// TwinCAT 3 PLC project RK_PapestraatV01
// ProgramVersion: 3.1.4024.12
// libraries:
//   Tc2_Standard, * (Beckhoff Automation GmbH)
//   Tc2_System, * (Beckhoff Automation GmbH)
//   Tc3_Module, * (Beckhoff Automation GmbH)
//   VisuSymbols,3.5.10.0,System
// project tree:
//   / GlobalTextList.TcGTLO, PlcTask.TcTTO, Visualization Manager.TcVMO (not stored)
//   GVLs/ GVL.TcGVL
//   POUs/ fbLightControl.TcPOU, fbLightControlV2.TcPOU, fbLightControl_ButtonAndDetect.TcPOU, fbVerwarming.TcPOU, MAIN.TcPOU, SturingVerwarming.TcPOU
//   VISUs/ InitSoftware.TcVIS
// real-time tasks:
//   TASK PlcTask: cycle T#10ms, priority 20, ADS port 350
// I/O:
//   DEVICE Device 2 (EtherCAT), AmsNetId 5.83.127.149.3.1
//     Term 8 (EK1200) [EK1200-5000 EtherCAT Power supply (2A E-Bus)]
//       Term 7 (EL1809) [EL1809 16Ch. Dig. Input 24V, 3ms]
//       Term 8 (EL1809) [EL1809 16Ch. Dig. Input 24V, 3ms]
//       Term 9 (EL2809) [EL2809 16Ch. Dig. Output 24V, 0.5A]
//       Term 10 (EL1859) [EL1859 8Ch. Dig. Input 24V, 3ms, 8Ch. Dig. Output 24V, 0.5A]
//       Term 11 (EL1008) [EL1008 8Ch. Dig. Input 24V, 3ms]
//       Term 14 (EL2008) [EL2008 8Ch. Dig. Output 24V, 0.5A]
//       Term 15 (EL9011) [EL9011 End Terminal]
// variable links:
//   RK-PapestraatV01/RK-PapestraatV01 Instance <-> Device 2 (EtherCAT)/Term 8 (EK1200)/Term 10 (EL1859)
//     PlcTask Inputs/GVL.I_Input{32..39} <-> Channel {1..8}/Input  (8 links)
//     PlcTask Outputs/GVL.Q_Light{16..19} <-> Channel {9..12}/Output  (4 links)
//     PlcTask Outputs/SturingVerwarming.bBranderAan <-> Channel 13/Output
//     PlcTask Outputs/SturingVerwarming.bKlepBureau <-> Channel 16/Output
//     PlcTask Outputs/SturingVerwarming.bKlepGroteZaal <-> Channel 14/Output
//     PlcTask Outputs/SturingVerwarming.bKlepKleineZaal <-> Channel 15/Output
//   RK-PapestraatV01/RK-PapestraatV01 Instance <-> Device 2 (EtherCAT)/Term 8 (EK1200)/Term 11 (EL1008)
//     PlcTask Inputs/SturingVerwarming.bDrukknopBureau <-> Channel 5/Input
//     PlcTask Inputs/SturingVerwarming.bDrukknopGroteZaal <-> Channel 1/Input
//     PlcTask Inputs/SturingVerwarming.bDrukknopKleineZaal <-> Channel 3/Input
//   RK-PapestraatV01/RK-PapestraatV01 Instance <-> Device 2 (EtherCAT)/Term 8 (EK1200)/Term 14 (EL2008)
//     PlcTask Outputs/SturingVerwarming.bKlepBureau <-> Channel 5/Output
//     PlcTask Outputs/SturingVerwarming.bKlepGroteZaal <-> Channel 1/Output
//     PlcTask Outputs/SturingVerwarming.bKlepKleineZaal <-> Channel 3/Output
//   RK-PapestraatV01/RK-PapestraatV01 Instance <-> Device 2 (EtherCAT)/Term 8 (EK1200)/Term 7 (EL1809)
//     PlcTask Inputs/GVL.I_Input01 <-> Channel 2/Input
//     PlcTask Inputs/GVL.I_Input02 <-> Channel 3/Input
//     PlcTask Inputs/GVL.I_Input03 <-> Channel 4/Input
//     PlcTask Inputs/GVL.I_Input04 <-> Channel 5/Input
//     PlcTask Inputs/GVL.I_Input05 <-> Channel 6/Input
//     PlcTask Inputs/GVL.I_Input06 <-> Channel 7/Input
//     PlcTask Inputs/GVL.I_Input08 <-> Channel 9/Input
//     PlcTask Inputs/GVL.I_Input09 <-> Channel 10/Input
//     PlcTask Inputs/GVL.I_Input10 <-> Channel 11/Input
//     PlcTask Inputs/GVL.I_Input11 <-> Channel 12/Input
//     PlcTask Inputs/GVL.I_Input12 <-> Channel 13/Input
//     PlcTask Inputs/GVL.I_Input13 <-> Channel 14/Input
//     PlcTask Inputs/GVL.I_Input14 <-> Channel 15/Input
//     PlcTask Inputs/GVL.I_Input15 <-> Channel 16/Input
//     PlcTask Inputs/SturingVerwarming.bThermostaatBureau <-> Channel 1/Input
//     PlcTask Inputs/SturingVerwarming.bThermostaatGroteZaal <-> Channel 8/Input
//   RK-PapestraatV01/RK-PapestraatV01 Instance <-> Device 2 (EtherCAT)/Term 8 (EK1200)/Term 8 (EL1809)
//     PlcTask Inputs/GVL.I_Input16 <-> Channel 1/Input
//     PlcTask Inputs/GVL.I_Input17 <-> Channel 2/Input
//     PlcTask Inputs/GVL.I_Input18 <-> Channel 3/Input
//     PlcTask Inputs/GVL.I_Input19 <-> Channel 4/Input
//     PlcTask Inputs/GVL.I_Input21 <-> Channel 6/Input
//     PlcTask Inputs/GVL.I_Input22 <-> Channel 7/Input
//     PlcTask Inputs/GVL.I_Input23 <-> Channel 8/Input
//     PlcTask Inputs/GVL.I_Input24 <-> Channel 9/Input
//     PlcTask Inputs/GVL.I_Input25 <-> Channel 10/Input
//     PlcTask Inputs/GVL.I_Input26 <-> Channel 11/Input
//     PlcTask Inputs/GVL.I_Input27 <-> Channel 12/Input
//     PlcTask Inputs/GVL.I_Input28 <-> Channel 13/Input
//     PlcTask Inputs/GVL.I_Input29 <-> Channel 14/Input
//     PlcTask Inputs/GVL.I_Input30 <-> Channel 15/Input
//     PlcTask Inputs/GVL.I_Input31 <-> Channel 16/Input
//     PlcTask Inputs/SturingVerwarming.bThermostaatKleineZaal <-> Channel 5/Input
//   RK-PapestraatV01/RK-PapestraatV01 Instance <-> Device 2 (EtherCAT)/Term 8 (EK1200)/Term 9 (EL2809)
//     PlcTask Outputs/GVL.Q_Light00 <-> Channel 1/Output
//     PlcTask Outputs/GVL.Q_Light01 <-> Channel 2/Output
//     PlcTask Outputs/GVL.Q_Light02 <-> Channel 3/Output
//     PlcTask Outputs/GVL.Q_Light03 <-> Channel 4/Output
//     PlcTask Outputs/GVL.Q_Light04 <-> Channel 5/Output
//     PlcTask Outputs/GVL.Q_Light05 <-> Channel 6/Output
//     PlcTask Outputs/GVL.Q_Light06 <-> Channel 7/Output
//     PlcTask Outputs/GVL.Q_Light07 <-> Channel 8/Output
//     PlcTask Outputs/GVL.Q_Light08 <-> Channel 9/Output
//     PlcTask Outputs/GVL.Q_Light09 <-> Channel 10/Output
//     PlcTask Outputs/GVL.Q_Light10 <-> Channel 11/Output
//     PlcTask Outputs/GVL.Q_Light11 <-> Channel 12/Output
//     PlcTask Outputs/GVL.Q_Light12 <-> Channel 13/Output
//     PlcTask Outputs/GVL.Q_Light13 <-> Channel 14/Output
//     PlcTask Outputs/GVL.Q_Light14 <-> Channel 15/Output
//     PlcTask Outputs/GVL.Q_Light15 <-> Channel 16/Output

CONFIGURATION RK_PapestraatV01
    RESOURCE PLC ON TwinCAT3
        TASK PlcTask(INTERVAL := T#10ms, PRIORITY := 20);
        PROGRAM MAIN WITH PlcTask : MAIN;
    END_RESOURCE
END_CONFIGURATION

// ---- GVLs/GVL.TcGVL
{attribute 'qualified_only'}
VAR_GLOBAL
	I_Input00		AT %I* :BOOL; // Thermostaat Bureau
	I_Input01		AT %I* :BOOL; // Ingang Bureau
	I_Input02		AT %I* :BOOL; // ingang Lesruimte Rechts
	I_Input03		AT %I* :BOOL; // ingang Lesruimte Links
	I_Input04		AT %I* :BOOL; // Voorbereiding knop uitgang
	I_Input05		AT %I* :BOOL; // Gang GarageZijde
	I_Input06		AT %I* :BOOL; // Knop Aan Trap (nog te ontdubbelen
	I_Input07		AT %I* :BOOL; // Thermostaat lesruimte
	I_Input08		AT %I* :BOOL; // lesruimte naar garage
	I_Input09		AT %I* :BOOL; // WC midden
	I_Input10		AT %I* :BOOL; // WC naast Tech
	I_Input11		AT %I* :BOOL; // Gang 1
	I_Input12		AT %I* :BOOL; // Gang 2
	I_Input13		AT %I* :BOOL; // Grote WC
	I_Input14		AT %I* :BOOL; // Tech Ruimte 
	I_Input15		AT %I* :BOOL; // opleidingslokaal rechts voorraan

	I_Input16		AT %I* :BOOL; // Lesruimte naar buiten
	I_Input17		AT %I* :BOOL; // AllesUitVoordeur
	I_Input18		AT %I* :BOOL; // 2de schakelaar opleidinslokaal deur naar berging
	I_Input19		AT %I* :BOOL; // Grime Grote WC
	I_Input20		AT %I* :BOOL; // Thermostaat vergader 
	I_Input21		AT %I* :BOOL; // c vergaderzaal
	I_Input22		AT %I* :BOOL; // Vergaderzaal DeurNaarBuiten 
	I_Input23		AT %I* :BOOL; // X Keuken
	I_Input24		AT %I* :BOOL; // Alles Uit 
	I_Input25		AT %I* :BOOL; // Garagezonder Deur Onderlinks
	I_Input26		AT %I* :BOOL; // Garagezonder Deur OnderRechts
	I_Input27		AT %I* :BOOL; // Poort 2 DeurDicht
	I_Input28		AT %I* :BOOL; // Poort 2 DeurOpen (Niet gebruikt)
	I_Input29		AT %I* :BOOL; // Poort 1 DeurDicht 
	I_Input30		AT %I* :BOOL; // Poort 1 DeurOpen (Niet Gebruikt)
	I_Input31		AT %I* :BOOL; // I ( opleiding deur naar buiten

	I_Input32		AT %I* :BOOL; // Garage drukknop
	I_Input33		AT %I* :BOOL; // Garage Drukknop2
	I_Input34		AT %I* :BOOL; // Verdieping 1 druknop 2
	I_Input35		AT %I* :BOOL; // AllesUit
	I_Input36		AT %I* :BOOL; // 
	I_Input37		AT %I* :BOOL;
	I_Input38		AT %I* :BOOL;
	I_Input39		AT %I* :BOOL;
	
//output values
	Q_Light00		AT %Q* :BOOL;	// Groot WC
	Q_Light01		AT %Q* :BOOL;	// Midden WC
	Q_Light02		AT %Q* :BOOL;   // Keuken
	Q_Light03		AT %Q* :BOOL;	// Buitenlicht achter
	Q_Light04		AT %Q* :BOOL;	// WC naast Tech Ruimte 
	Q_Light05		AT %Q* :BOOL;  	// vergaderzaal
	Q_Light06		AT %Q* :BOOL;  	// bureau
	Q_Light07		AT %Q* :BOOL;  	// Lesruimte deel 1
	Q_Light08		AT %Q* :BOOL;  	// Garage Deur	
	Q_Light09		AT %Q* :BOOL;	// Garage enkel poort
	Q_Light10		AT %Q* :BOOL; 	// Verdiep 1 trap
	Q_Light11		AT %Q* :BOOL; 	// verdiep 1 ver
	Q_Light12		AT %Q* :BOOL;	// Berg Ruimte 
	Q_Light13		AT %Q* :BOOL;	// Gang Deel 2
	Q_Light14		AT %Q* :BOOL;	// GrimeLicht grote WC
	Q_Light15		AT %Q* :BOOL;	// Tech Ruimte
	
	Q_Light16		AT %Q* :BOOL;	// IndicatieLicht DeurGarage
	Q_Light17		AT %Q* :BOOL; 	// Lesruimte Deel 2
	Q_Light18		AT %Q* :BOOL; 	//
	Q_Light19		AT %Q* :BOOL;	// Lichtje GarageZonderDeur
	Q_Light20		AT %Q* :BOOL;	// Verwarming 1
	Q_Light21		AT %Q* :BOOL;	// Verwarming 2
	Q_Light22		AT %Q* :BOOL;	// Verwarming 3
	Q_Light23		AT %Q* :BOOL;	// Verwarming 4 
	
	
	LesruimteLichtAan		:BOOL;
	BureauLichtAan			:BOOL;
	Vergaderzaal			:BOOL;
	
// placeholder values
	I_Inputxx		AT %I* :BOOL;
	Q_LightXX		AT %Q* :BOOL;
	
	//I_Temp01		AT %I* :BOOL;
	//I_Temp02		AT %I* :BOOL;
	//I_Temp03		AT %I* :BOOL;
	//I_Temp04		AT %I* :BOOL;

	
END_VAR

// ---- POUs/MAIN.TcPOU
PROGRAM MAIN
VAR
	cnt			: UINT;
	
	fbLight00		: fbLightControl;
	fbLight01		: fbLightControl;
	fbLight02		: fbLightControl;
	fbLight03		: fbLightControl;
	fbLight04		: fbLightControl;
	fbLight05		: fbLightControl; // testje
	fbLight06		: fbLightControl;
	fbLight07		: fbLightControlV2;
	fbLight08		: fbLightControl_ButtonAndDetect;
	fbLight09		: fbLightControl;
	fbLight10		: fbLightControl;
	fbLight11		: fbLightControl;
	fbLight12		: fbLightControl;
	fbLight13		: fbLightControl;
	fbLight14		: fbLightControl;
//	fbLight15		: fbLightControl;
	
	bOutputActief	: BOOL;
	
	bForceOff		:BOOL;
	bForceOn		:BOOL;
	
	InputTriggerAllesUit		: R_trig; 
	
	LesruimteLichtAan: INT;
END_VAR

 cnt := cnt +1;



InputTriggerAllesUit(CLK := GVL.I_Input35 OR GVL.I_Input24 OR gvl.I_Input17);
	
// Actual light control

fbLight00(bButton:= GVL.I_Input32 , 
			bForceOff:= InputTriggerAllesUit.Q, 
			bForceOn:= , 
			bLight=> gvl.Q_Light07,
			bLight=> gvl.Q_Light04,
			);
// Grote WC hoofdlicht

GVL.Q_Light01 := GVL.I_Input09; //midden WC
GVL.Q_Light00 := GVL.I_Input13; // Grote WC 
GVL.Q_Light04 := GVL.I_Input10;// WC naast tech
GVL.Q_Light15 := GVL.I_Input14; // tech ruimte
GVL.Q_Light12 := GVL.I_Input08;// BergRuimte =Detector
GVL.Q_Light13 := GVL.I_Input11 OR GVL.I_Input12;// Gang deel2 detector


//verlichting Bureau
		


		

		
		// Licht Keuken
fbLight02(bButton:= GVL.I_Input03 OR GVL.I_Input23 ,  // check other button 
			bForceOff:= InputTriggerAllesUit.Q, 
			bForceOn:= , 
			bLight=> gvl.Q_Light02,
		);
		
// Licht Buiten	
fbLight03(bButton:= GVL.I_Input04 OR GVL.I_Input31 OR GVL.I_Input22, 
			bForceOff:= InputTriggerAllesUit.Q, 
			bForceOn:= , 
			bLight=> gvl.Q_Light03,
		);
		
// 	vergaderzaal

fbLight05(bButton:= GVL.I_Input21, 
			bForceOff:= InputTriggerAllesUit.Q, 
			bForceOn:= , 
			bLight=> gvl.Q_Light05
		);	
// Bureau

fbLight06(bButton:= GVL.I_Input01,
			bForceOff:= InputTriggerAllesUit.Q, 
			bForceOn:= , 
			
			bLight=> gvl.Q_Light06
		);	
// Lesruimte 	
fbLight07(bButtonhoofdFunctie:= GVL.I_Input02 OR GVL.I_Input15 ,
			bButton2 := GVL.I_Input18 OR GVL.I_Input16, // 16 should move to outside
			bForceOff:= InputTriggerAllesUit.Q, 
			bForceOn:= , 
			bLight1=> gvl.Q_Light07,
			bLight2=> gvl.Q_Light17
		);	
// Garage 	
fbLight08(bButton:= GVL.I_Input33 OR GVL.I_Input05 OR GVL.I_Input32 OR GVL.I_Input26,
			bDetection := GVL.I_Input37  ,
			bDeurDetectie :=  NOT(GVL.I_Input29) OR NOT(GVL.I_Input27),
			bForceOff:= InputTriggerAllesUit.Q, 
			bForceOn:= , 
			bInhibit:= InputTriggerAllesUit.Q, 
			bLight=> gvl.Q_Light08,
			bLight=> gvl.Q_Light09,
		);
// Deze knop laat toe om de detectie over te nemen 
// Logica nog te verbeteren met de alles uit samen te werken


(*TODO: remove after logic validation
gvl.Q_Light08 := gvl.Q_Light08 OR GVL.I_Input37;
gvl.Q_Light09 := gvl.Q_Light09 OR GVL.I_Input37;*)

// zaal boven
fbLight10(bButton:= GVL.I_Input34 OR GVL.I_Input06 OR GVL.I_Input25, 
			bForceOff:= InputTriggerAllesUit.Q, 
			bForceOn:= , 
			bLight=> gvl.Q_Light10,
			bLight=> gvl.Q_Light11
			);

// GrimeLicht Grote WC
fbLight14(bButton:= GVL.I_Input19 , 
			bForceOff:= InputTriggerAllesUit.Q, 
			bForceOn:= , 
			bLight=> gvl.Q_Light14
		);	

		
bOutputActief := fbLight00.bLight
				OR fbLight01.bLight
				OR fbLight02.bLight
				OR fbLight03.bLight
				OR fbLight04.bLight
				OR fbLight05.bLight
				OR fbLight06.bLight
				OR fbLight07.bLight1 OR fbLight07.bLight2
				OR fbLight08.bLight
				OR fbLight09.bLight
				OR fbLight10.bLight
				OR fbLight11.bLight
				OR fbLight12.bLight
				OR fbLight13.bLight
				OR fbLight14.bLight;

GVL.Q_Light16 :=  bOutputActief;				

// Activeer Verwarming

	GVL.LesruimteLichtAan := gvl.Q_Light07 OR gvl.Q_Light17 OR gvl.Q_Light02;
	GVL.BureauLichtAan	  := gvl.Q_Light06 ;
	GVL.Vergaderzaal	  := gvl.Q_Light05 ;

SturingVerwarming();

END_PROGRAM

// ---- POUs/fbLightControl.TcPOU
FUNCTION_BLOCK fbLightControl
		
VAR_INPUT
	bButton				: BOOL;
	bForceOff			: BOOL;
	bForceOn			: BOOL;

END_VAR
VAR_OUTPUT
	bLight				: BOOL;
	
END_VAR
VAR
	InputTrigger		: R_trig; 

	
END_VAR

// This is the first version, ignoring all debounce timers and other issues 
// Base function is a to allow switching a light on and of and having a general reset and general on ( used for construcion)

InputTrigger(CLK :=  bButton);

IF InputTrigger.Q THEN
	
	bLight := NOT(bLight);

END_IF

// Deze functie zorgt voor alles aan/Uit Functionaliteit
IF bForceOff THEN
	bLight := FALSE;
END_IF

IF bForceOn THEN
	bLight := TRUE;
END_IF

(*function notes: long klick functionality not added, most likley this will be part of another function
This could be a dedicated filter function linked to these functions as needed
*)

END_FUNCTION_BLOCK

// ---- POUs/fbLightControlV2.TcPOU
FUNCTION_BLOCK fbLightControlV2
		
VAR_INPUT
	bButtonhoofdFunctie				: BOOL;
	bButton2				: BOOL;
	bForceOff			: BOOL;
	bForceOn			: BOOL;

END_VAR
VAR_OUTPUT
	bLight1				: BOOL;
	bLight2				: BOOL;	
	
END_VAR
VAR
	InputTriggerHoofd		: R_trig; 
	InputTrigger2		: R_trig; 
	test:BOOL;
	iCaseVar			:UINT; 
	

	
END_VAR


// This is the first version, ignoring all debounce timers and other issues 
// Base function is a to allow switching a light on and of and having a general reset and general on ( used for construcion)

InputTriggerHoofd(CLK :=  bButtonhoofdFunctie);
InputTrigger2(CLK :=  bButton2);


IF InputTriggerHoofd.Q THEN
	
// ALs alles uit, dan alles aan
	IF (iCaseVar = 0) THEN
		iCaseVar := 1;
	ELSE
		iCaseVar := 0;
	END_IF
END_IF 

IF InputTrigger2.Q THEN
	
	// ALs alles aan, dan de voorste lichten uit
	IF (iCaseVar = 1) THEN
		iCaseVar := 2;
	ELSIF (iCaseVar = 2) THEN
		iCaseVar := 1;
	END_IF
	
END_IF

CASE iCaseVar OF
0:
    bLight1 := FALSE;
	bLight2 := FALSE;
1:
    bLight1 := TRUE;
	bLight2 := TRUE;	
2:
    bLight1 := TRUE;
	bLight2 := FALSE;
3: // eigenlijk niet noodzakelijk
	iCaseVar := 0;
ELSE
	iCaseVar := 0;
END_CASE;




// Deze functie zorgt voor alles aan/Uit Functionaliteit
IF bForceOff THEN
	iCaseVar := 0;
END_IF

IF bForceOn THEN
	iCaseVar := 1;
END_IF

(*function notes: long klick functionality not added, most likley this will be part of another function
This could be a dedicated filter function linked to these functions as needed
*)

END_FUNCTION_BLOCK

// ---- POUs/fbLightControl_ButtonAndDetect.TcPOU
FUNCTION_BLOCK fbLightControl_ButtonAndDetect
		
VAR_INPUT
	bButton				: BOOL;
	bDeurDetectie		: BOOL;
	bForceOff			: BOOL;
	bForceOn			: BOOL;
	bDetection			: BOOL;
	bInhibit			:BOOL;
	
	//tInhibitTime		:TIME := T#60s;
    tDeurOpenTime		:TIME := T#10m;
END_VAR
VAR_OUTPUT
	bLight				: BOOL;
	
END_VAR
VAR
	InputTrigger		: R_trig; 
	DetectieTrigger		: R_trig; 
	DeurTrigger			: R_trig; 
	//TimerInhibit		: TOF; 
	TimerDeurdetectie	: TON;
	bInternLichtVarKnop : BOOL;
	bOverneemDeurDetectie :BOOL;
	
END_VAR

// This is the first version, ignoring all debounce timers and other issues 
// Base function is a to allow switching a light on and of and having a general reset and general on ( used for construcion)

//Button detection
InputTrigger(CLK :=  bButton);

//rising edge detection used for the optical detection and deur detection
DetectieTrigger(clk := bDetection);
DeurTrigger(clk := bDeurDetectie);
// button function
IF InputTrigger.Q THEN
	
	IF bInternLichtVarKnop OR bOverneemDeurDetectie THEN
		bOverneemDeurDetectie :=  FALSE;
	END_IF
	bInternLichtVarKnop := NOT(bInternLichtVarKnop);

END_IF

// Dit onderdeel triggert als de deur opent en blijft de ingestelde tijd lopen na het sleuiten

IF DetectieTrigger.Q OR DeurTrigger.Q THEN 
	bOverneemDeurDetectie := TRUE;
END_IF

TimerDeurdetectie(In := bOverneemDeurDetectie AND(NOT(DetectieTrigger.Q )), PT:= tDeurOpenTime);


IF TimerDeurdetectie.Q THEN
	bOverneemDeurDetectie := FALSE;
END_IF

// Deze functie zorgt voor alles aan/Uit Functionaliteit
IF bForceOff THEN
	bInternLichtVarKnop := FALSE;
	bOverneemDeurDetectie := FALSE;
END_IF

IF bForceOn THEN
	bInternLichtVarKnop := TRUE;
END_IF


bLight := (bInternLichtVarKnop OR  bOverneemDeurDetectie) ;




(*function notes: long klick functionality not added, most likley this will be part of another function
This could be a dedicated filter function linked to these functions as needed
*)

END_FUNCTION_BLOCK

// ---- POUs/SturingVerwarming.TcPOU
PROGRAM SturingVerwarming
VAR
	fbGroteVergaderzaal					:fbVerwarming;
	fbKleineVergaderzaal				:fbVerwarming;
	fbBureau							:fbVerwarming;
	
	bDrukknopGroteZaal			AT %I*		:BOOL; //Drukknoppen te voorzien op kast
	bDrukknopKleineZaal			AT %I*		:BOOL; //Drukknoppen te voorzien op kast
	bDrukknopBureau				AT %I*		:BOOL; //Drukknoppen te voorzien op kast
	
	bThermostaatGroteZaal		AT %I*		:BOOL; 
	bThermostaatKleineZaal		AT %I*		:BOOL;
	bThermostaatBureau			AT %I*		:BOOL;
	
	bKlepGroteZaal				AT %Q*		:BOOL; //Uitgangen naar relais in kastje aan brander
	bKlepKleineZaal				AT %Q*		:BOOL; //Uitgangen naar relais in kastje aan brander
	bKlepBureau					AT %Q*		:BOOL;	//Uitgangen naar relais in kastje aan brander
	bBranderAan					AT %Q*		:BOOL; //Uitgangen naar relais in kastje aan brander
	
	
	// tTijdVoorStart is de tijd dat de verwarming aangaat nadat iemand op de knop druk, die op de kast voorzien is.
	
END_VAR

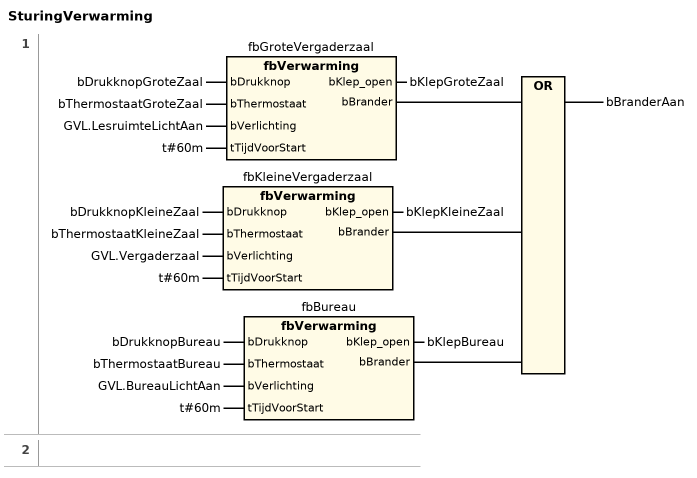
// NETWORK 1
fbGroteVergaderzaal(
    bDrukknop := bDrukknopGroteZaal,
    bThermostaat := bThermostaatGroteZaal,
    bVerlichting := GVL.LesruimteLichtAan,
    tTijdVoorStart := t#60m,
    bKlep_open => bKlepGroteZaal); // fbVerwarming
fbKleineVergaderzaal(
    bDrukknop := bDrukknopKleineZaal,
    bThermostaat := bThermostaatKleineZaal,
    bVerlichting := GVL.Vergaderzaal,
    tTijdVoorStart := t#60m,
    bKlep_open => bKlepKleineZaal); // fbVerwarming
fbBureau(
    bDrukknop := bDrukknopBureau,
    bThermostaat := bThermostaatBureau,
    bVerlichting := GVL.BureauLichtAan,
    tTijdVoorStart := t#60m,
    bKlep_open => bKlepBureau); // fbVerwarming
bBranderAan := fbGroteVergaderzaal.bBrander OR fbKleineVergaderzaal.bBrander OR fbBureau.bBrander;

// NETWORK 2

END_PROGRAM

// ---- POUs/fbVerwarming.TcPOU
FUNCTION_BLOCK fbVerwarming
VAR_INPUT
	bDrukknop				:BOOL;
	bThermostaat			:BOOL;
	bVerlichting			:BOOL;
	tTijdVoorStart			:TIME;
END_VAR
VAR_OUTPUT
	bKlep_open				:BOOL;
	bBrander				:BOOL;
END_VAR
VAR
	bUitlooptijdKlep			:BOOL;
	Uitlooptijd					:tof;
	TijdsduurVoorverwarming		:tof;
	Brander						:F_TRIG;
	
END_VAR

TijdsduurVoorverwarming(IN:= bDrukknop, PT:= tTijdVoorStart, Q=> , ET=> );

Uitlooptijd(IN:= bUitlooptijdKlep, PT:= T#30S, Q=> , ET=> );

IF Uitlooptijd.Q THEN
	bKlep_open := TRUE;
	ELSE
	bKlep_open := FALSE;
	END_IF

IF (TijdsduurVoorverwarming.Q OR bVerlichting) AND bThermostaat THEN
		bUitlooptijdKlep := TRUE;
		bBrander := TRUE;
		ELSE
		bUitlooptijdKlep :=FALSE;
		bBrander := FALSE;
END_IF

END_FUNCTION_BLOCK

// ---- GlobalTextList.TcGTLO
TEXTLIST GlobalTextList
  985 = 'input 0- 7'
  530 = 'input 16-23'
  799 = 'input 24-31'
  262 = 'input 8-15'
END_TEXTLIST

// ---- VISUs/InitSoftware.TcVIS
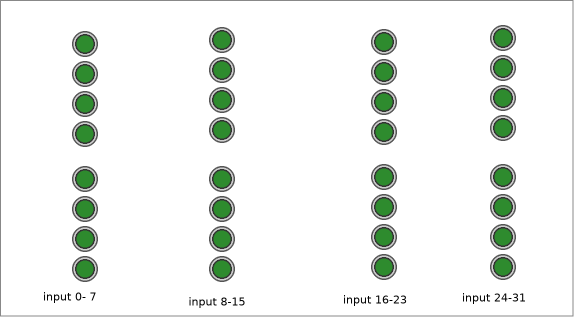
VISUALIZATION InitSoftware  // 574x317
    Lamp1 (69,29 32x30), variable: GVL.I_Input00, style: Lamp-Lamp1-Green
    Lamp1 (69,59 32x30), variable: GVL.I_Input01, style: Lamp-Lamp1-Green
    Lamp1 (69,89 32x30), variable: GVL.I_Input02, style: Lamp-Lamp1-Green
    Lamp1 (69,119 32x30), variable: GVL.I_Input03, style: Lamp-Lamp1-Green
    Lamp1 (69,164 32x30), variable: GVL.I_Input04, style: Lamp-Lamp1-Green
    Lamp1 (69,194 32x30), variable: GVL.I_Input05, style: Lamp-Lamp1-Green
    Lamp1 (69,224 32x30), variable: GVL.I_Input06, style: Lamp-Lamp1-Green
    Lamp1 (69,254 32x30), variable: GVL.I_Input07, style: Lamp-Lamp1-Green
    Lamp1 (206,25 32x30), variable: GVL.I_Input08, style: Lamp-Lamp1-Green
    Lamp1 (206,55 32x30), variable: GVL.I_Input09, style: Lamp-Lamp1-Green
    Lamp1 (206,85 32x30), variable: GVL.I_Input10, style: Lamp-Lamp1-Green
    Lamp1 (206,115 32x30), variable: GVL.I_Input11, style: Lamp-Lamp1-Green
    Lamp1 (206,164 32x30), variable: GVL.I_Input12, style: Lamp-Lamp1-Green
    Lamp1 (206,194 32x30), variable: GVL.I_Input13, style: Lamp-Lamp1-Green
    Lamp1 (206,224 32x30), variable: GVL.I_Input14, style: Lamp-Lamp1-Green
    Lamp1 (206,254 32x30), variable: GVL.I_Input15, style: Lamp-Lamp1-Green
    Lamp1 (368,27 32x30), variable: GVL.I_Input16, style: Lamp-Lamp1-Green
    Lamp1 (368,57 32x30), variable: GVL.I_Input17, style: Lamp-Lamp1-Green
    Lamp1 (368,87 32x30), variable: GVL.I_Input18, style: Lamp-Lamp1-Green
    Lamp1 (368,117 32x30), variable: GVL.I_Input19, style: Lamp-Lamp1-Green
    Lamp1 (368,162 32x30), variable: GVL.I_Input20, style: Lamp-Lamp1-Green
    Lamp1 (368,192 32x30), variable: GVL.I_Input21, style: Lamp-Lamp1-Green
    Lamp1 (368,222 32x30), variable: GVL.I_Input22, style: Lamp-Lamp1-Green
    Lamp1 (368,252 32x30), variable: GVL.I_Input23, style: Lamp-Lamp1-Green
    Lamp1 (487,23 32x30), variable: GVL.I_Input24, style: Lamp-Lamp1-Green
    Lamp1 (487,53 32x30), variable: GVL.I_Input25, style: Lamp-Lamp1-Green
    Lamp1 (487,83 32x30), variable: GVL.I_Input26, style: Lamp-Lamp1-Green
    Lamp1 (487,113 32x30), variable: GVL.I_Input27, style: Lamp-Lamp1-Green
    Lamp1 (487,162 32x30), variable: GVL.I_Input28, style: Lamp-Lamp1-Green
    Lamp1 (487,192 32x30), variable: GVL.I_Input29, style: Lamp-Lamp1-Green
    Lamp1 (487,222 32x30), variable: GVL.I_Input30, style: Lamp-Lamp1-Green
    Lamp1 (487,252 32x30), variable: GVL.I_Input31, style: Lamp-Lamp1-Green
    Label (-5,282 150x30), "input 0- 7"
    Label (300,285 150x30), "input 16-23"
    Label (142,287 150x30), "input 8-15"
    Label (419,283 150x30), "input 24-31"
END_VISUALIZATION
